// TIA Portal V18 export
TYPE "DI"
// stored: IsFailsafeCompliant false
   STRUCT
      START : Bool;
      STOP : Bool;
      EMERGENCY : Bool;
      ACKNOWLEDGE : Bool;
      "AUTO/MANUAL" : Bool;
      "RECUPARATION TANK HL" : Bool;
      "RECUPARATION TANK LL" : Bool;
      "HOT WATER TANK HL" : Bool;
      "HOT WATER TANK LL" : Bool;
      "CAUSTIC TANK HL" : Bool;
      "CAUSTIC TANK LL" : Bool;
      "ACID TANK HL" : Bool;
      "ACID TANK LL" : Bool;
      "SUPPLY PUMP RUN (VFD)" : Bool;
      RESERVED : Bool;
      RESERVED_1 : Bool;
      "SUPPLY PUMP TRIP (VFD)" : Bool;
      "ACID DOSING PUMP RUN" : Bool;
      "ACID DOSING PUMP TRIP" : Bool;
      "CAUSTIC DOSING PUMP RUN" : Bool;
      "CAUSTIC DOSING PUMP TRIP" : Bool;
      "RETURN PUMP 1 RUN" : Bool;
      "RETURN PUMP 1 TRIP" : Bool;
      "RETURN PUMP 2 RUN" : Bool;
      "RETURN PUMP 2 TRIP" : Bool;
      "RETURN PUMP 3 RUN" : Bool;
      "RETURN PUMP 3 TRIP" : Bool;
      "FLOW SWITCH" : Bool;
      "PRESSURE SWITCH" : Bool;
      SPARE_1 : Bool;
      SPARE_2 : Bool;
      SPARE_3 : Bool;
   END_STRUCT;
END_TYPE
